FUNCTION_BLOCK FB_DeviceMonitor

VAR_IN_OUT
//	devices : ARRAY[*] OF FB_MonitoredDevice;
//	Devices : ARRAY[*] OF MonitoredDeviceStruct;
END_VAR

VAR
	devices : FB_BA_DynamicArray;
END_VAR

//devices.uiEntrySize := 50;

METHOD AddMonitoredDevice : BOOL // Returns the monitored device instance that has just been added
VAR_INPUT
	device : FB_MonitoredDevice;
//	name : WSTRING(255);
//	location : WSTRING(255);
//	description : WSTRING(255);
END_VAR

VAR
//	uNewMaxIndex : DINT;
//	fbMonitoredDevice : FB_MonitoredDevice;
//	stMonitoredDevice : ST_MonitoredDevice;
	resultIndex: DINT;
END_VAR
// Find the current max index in the existing array
//uNewMaxIndex := UPPER_BOUND(devices,1);

// Create a new monitored device instance
//fbMonitoredDevice.device := device.pValue;
//fbMonitoredDevice.deviceId := devices.diCount;
//device.deviceId := uNewMaxIndex;
//device.deviceId := devices.diCount;
device.deviceId := devices.LastIndex;

//fbMonitoredDevice.name := name;
//fbMonitoredDevice.location := location;
//fbMonitoredDevice.description := description;

devices.AddEntryPtr(pEntry := ADR(device));

// Populate the response struct with the instance and it's ID/index location
//stMonitoredDevice.device := fbMonitoredDevice;
//stMonitoredDevice.deviceId := uNewMaxIndex;

// Add the new device instance to the array of monitored devices
//Devices[uNewMaxIndex] := stMonitoredDevice;
//Devices[uNewMaxIndex] := fbMonitoredDevice;
//devices[uNewMaxIndex] := device;

// Return the response struct
//AddMonitoredDevice := stMonitoredDevice;
//AddMonitoredDevice := fbMonitoredDevice;
AddMonitoredDevice := TRUE;
END_METHOD

END_FUNCTION_BLOCK

(* stored: Version 1.1.0.1, ProductVersion 3.1.4024.11
   POU FB_DeviceMonitor: Id {bc1bc499-3913-423a-945b-98ef54d797c7}, SpecialFunc None
   Method AddMonitoredDevice: Id {3d226fca-917d-4593-a4df-24a17244406a} *)
